TYPE T_Ctrl_SIf_HFE_Cur :
STRUCT
END_STRUCT
END_TYPE

(* stored: Version 1.1.0.1, ProductVersion 3.1.0.23
   DUT T_Ctrl_SIf_HFE_Cur: Id {34db0434-8f77-47a8-9f61-1ab0eceee1c2} *)
